TYPE stEasyPumpsParamter :
STRUCT
 		xRdyCmd:BOOL;
		xStart:BOOL;
		xReset:BOOL;
		xBusy:BOOL;
		xError:BOOL;
		xDone:BOOL; 
		
		// 手动校准步骤
		iMCalibStep,iOldMCalibStep: INT;

 		iPumpContorller:INT;
		iPumpModule:INT;
		rSetVolume:REAL;
		rRunTime :REAL;
		iCycleNum:INT;
		iBackAngle:INT;
		rAverageRealVolume:REAL;
		arrRealVolume:ARRAY[1..3] OF REAL;
		arrTestRealVolume:ARRAY[1..50] OF REAL;
		arrRecordVolume:ARRAY[1..50] OF REAL;
		iInjectCounter:INT;
		iCalibCounter:INT;
		iRecordCounter:INT;
		//操作
		
		xModulePushStart:BOOL;//单通道注液开始
		xCalibTestStart:BOOL;//校准测试开始
		xRecordDataStart:BOOL;//记录数据开始
		xModulePushOK:BOOL;//注液OK
		xCalibTestOK:BOOL;//校准测试OK
		xRecordDataOK:BOOL;//记录数据OK
		tStableDelay: TON;
		xInitCalibration:BOOL;//初始化校准系数
		xGotoPosition:BOOL;//去校准位置
		xNeedInjectAgain:BOOL;//需要重新注液
		
		//上下偏差
		rESVolume: REAL;//上偏差
		rEIVolume: REAL;//下偏差
		
END_STRUCT
END_TYPE

(* stored: Version 1.1.0.1, ProductVersion 3.1.4024.9
   DUT stEasyPumpsParamter: Id {03770599-bb0d-430f-95ea-fb5139a79cb3} *)
